// TIA Portal V18 export
DATA_BLOCK "=S1+MA1-QQ1"   // DB21, F_DB
// stored: InstanceOfName 02_Safety_Door, InstanceOfType FB
"02_Safety_Door"
   // VAR_INPUT
   //    Bypass_For_Commissioning : Bool;
   //    DIAG : Bool;
   //    CH1 : Bool;
   //    CH2 : Bool;
   //    "Sorter_Running_from MSC" : Bool;
   //    Sorter_Stop_from_Encoder : Bool;
   //    Open_Request : Bool;
   //    Alarm_Filter : Bool;
   //    Sorter_Door : Bool;
   //    ACK_NEC : Bool;
   //    ACK : Bool;
   //    ON_Lamp : Bool;
   // END_VAR
   // VAR_OUTPUT
   //    Solenoid : Bool;
   //    EM_Cut : Bool;
   //    EM_Cut_Delay : Bool;
   //    Diag_Open : Bool;
   //    Diag_Alarm : Bool;
   //    Reset_Lamp : Bool;
   // END_VAR
   // VAR
   //    "E-STOP" : ESTOP1;
   //    TON_Alarm : TON;
   //    TOF_DoorLamp : TOF;
   // END_VAR
BEGIN
END_DATA_BLOCK
